{attribute 'qualified_only'}
{attribute 'strict'}
{attribute 'to_string'}
TYPE E_SL3K4State :
(
	TRANSITION := 0,
	NORMAL := 1,
	MAINTENANCE := 2
);
END_TYPE

(* stored: Version 1.1.0.1
   DUT E_SL3K4State: Id {5e8e7771-0770-435f-b3dd-c64a6cafa63b} *)
